FUNCTION_BLOCK PUBLIC EventEmitter_TestSuite EXTENDS TcUnit.FB_TestSuite
VAR
END_VAR

CheckEmitWorksWithHandler();
CheckEmitWorksWithMultipleHandlers();
CheckEventIsNotSentToTheWrongHandler();
CheckOffEventUnregistersAHandler();
CheckClearUnregistersMultipleHandlers();
CheckOnceEventCorrectlyCallsHandler();
CheckOnceEventCorrectlyCallsHandlerOnlyOnce();

METHOD PUBLIC CheckClearUnregistersMultipleHandlers
VAR
	mockEvent : MockEvent;
	mockHandler1 : MockEventHandler;
	mockHandler2 : MockEventHandler;
	eventEmitter : EventEmitter;
	eventReceived : BOOL;
END_VAR
TEST('CheckClearUnregistersMultipleHandlers');

eventEmitter.OnEvent('test', mockHandler1);
eventEmitter.OnEvent('test', mockHandler2);
eventEmitter.Clear();

eventEmitter.Emit('test',mockEvent);
eventReceived := mockHandler1.EqualsLastEvent(mockEvent) OR mockHandler2.EqualsLastEvent(mockEvent) ;

AssertFalse(
	Condition := eventReceived,
	Message := 'Event Emitter did not correctly unregister multiple handlers following a clear'
);

TEST_FINISHED();
END_METHOD

METHOD PUBLIC CheckEmitWorksWithHandler
VAR
	mockEvent : MockEvent;
	mockHandler : MockEventHandler;
	eventEmitter : EventEmitter;
	eventReceived : BOOL;
END_VAR
TEST('CheckEmitWorksWithHandler');

eventEmitter.OnEvent('test', mockHandler);

eventEmitter.Emit('test',mockEvent);
eventReceived := mockHandler.EqualsLastEvent(mockEvent);

AssertTrue(
	Condition := eventReceived,
	Message := 'Event Emitter did not correctly emmit the event to the handler'
);

TEST_FINISHED();
END_METHOD

METHOD PUBLIC CheckEmitWorksWithMultipleHandlers
VAR
	mockEvent : MockEvent;
	mockHandler1 : MockEventHandler;
	mockHandler2 : MockEventHandler;
	eventEmitter : EventEmitter;
	eventReceived : BOOL;
END_VAR
TEST('CheckEmitWorksWithMultipleHandlers');

eventEmitter.OnEvent('test', mockHandler1);
eventEmitter.OnEvent('test', mockHandler2);

eventEmitter.Emit('test',mockEvent);
eventReceived := mockHandler1.EqualsLastEvent(mockEvent) AND mockHandler2.EqualsLastEvent(mockEvent) ;

AssertTrue(
	Condition := eventReceived,
	Message := 'Event Emitter did not correctly emmit the event to multiple handlers'
);

TEST_FINISHED();
END_METHOD

METHOD PUBLIC CheckEventIsNotSentToTheWrongHandler
VAR
	mockEvent : MockEvent;
	mockHandler : MockEventHandler;
	eventEmitter : EventEmitter;
	eventReceived : BOOL;
END_VAR
TEST('CheckEventIsNotSentToTheWrongHandler');

eventEmitter.OnEvent('foo', mockHandler);

eventEmitter.Emit('bar',mockEvent);
eventReceived := mockHandler.EqualsLastEvent(mockEvent);

AssertFalse(
	Condition := eventReceived,
	Message := 'Event Emitter sent the event to the wrong handler'
);

TEST_FINISHED();
END_METHOD

METHOD PUBLIC CheckOffEventUnregistersAHandler
VAR
	mockEvent : MockEvent;
	mockHandler : MockEventHandler;
	eventEmitter : EventEmitter;
	eventReceived : BOOL;
END_VAR
TEST('CheckOffEventUnregistersAHandler');

eventEmitter.OnEvent('test', mockHandler);
eventEmitter.OffEvent('test', mockHandler);

eventEmitter.Emit('test',mockEvent);
eventReceived := mockHandler.EqualsLastEvent(mockEvent);

AssertFalse(
	Condition := eventReceived,
	Message := 'Event Emitter did not correctly unregister the event handler using the off method'
);

TEST_FINISHED();
END_METHOD

METHOD PUBLIC CheckOnceEventCorrectlyCallsHandler
VAR
	mockEvent : MockEvent;
	mockHandler : MockEventHandler;
	eventEmitter : EventEmitter;
	eventReceived : BOOL;
END_VAR
TEST('CheckOnceEventCorrectlyCallsHandler');

eventEmitter.OnceEvent('test', mockHandler);

eventEmitter.Emit('test',mockEvent);
eventReceived := mockHandler.EqualsLastEvent(mockEvent);

AssertTrue(
	Condition := eventReceived,
	Message := 'Event Emitter did not notify the handler'
);

TEST_FINISHED();
END_METHOD

METHOD PUBLIC CheckOnceEventCorrectlyCallsHandlerOnlyOnce
VAR
	mockEvent : MockEvent;
	mockHandler : MockEventHandler;
	eventEmitter : EventEmitter;
	eventCount : INT;
	expected : INT := 1;
END_VAR
TEST('CheckOnceEventCorrectlyCallsHandlerOnlyOnce');

eventEmitter.OnceEvent('test', mockHandler);

eventEmitter.Emit('test',mockEvent);
eventEmitter.Emit('test',mockEvent);
eventCount := mockHandler.EventsHandled;

AssertEquals(
	Expected := expected,
	Actual := eventCount,
	Message := 'Event Emitter notified the handler too many times'
);

TEST_FINISHED();
END_METHOD

END_FUNCTION_BLOCK

(* stored: Version 1.1.0.1, ProductVersion 3.1.4024.12
   POU EventEmitter_TestSuite: Id {c771dd79-b70b-0181-1b27-c5e2c81ee9a4}, SpecialFunc None
   Method CheckClearUnregistersMultipleHandlers: Id {6f968a81-0a57-03c6-3348-3b3f43b11e67}
   Method CheckEmitWorksWithHandler: Id {2e5817dc-28f3-0522-2aca-21ad8e95462f}
   Method CheckEmitWorksWithMultipleHandlers: Id {ca286491-29ce-0ee7-232d-791d78869866}
   Method CheckEventIsNotSentToTheWrongHandler: Id {c9d6842b-c5e0-0fa4-11db-eb3e4bccea3b}
   Method CheckOffEventUnregistersAHandler: Id {0291f32e-8068-0b28-38a8-cb83a2bc5dca}
   Method CheckOnceEventCorrectlyCallsHandler: Id {b82d80da-8d21-4c3f-b461-1bcdf25058fc}
   Method CheckOnceEventCorrectlyCallsHandlerOnlyOnce: Id {41e2f222-2d9a-4d62-b09f-7d10f71b8a0c} *)
